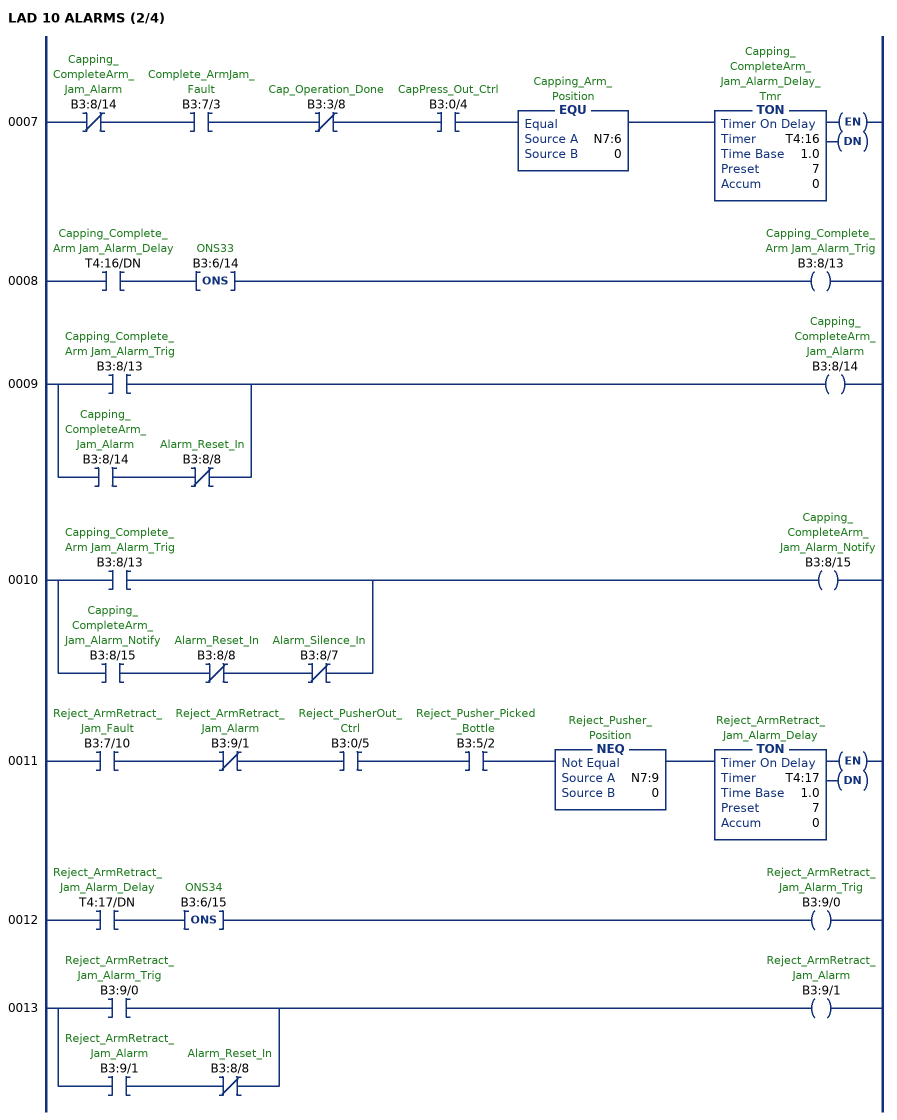
% Rung: 7 %
SOR XIO B3:8/14 XIC B3:7/3 XIO B3:3/8 XIC B3:0/4 EQU N7:6 0 TON T4:16 1.0 7 0 EOR
%   B3:8/14  "Capping_CompleteArm_ Jam_Alarm" %
%   B3:7/3  "Complete_ArmJam_ Fault" %
%   B3:3/8  "Cap_Operation_Done" %
%   B3:0/4  "CapPress_Out_Ctrl" %
%   N7:6  "Capping_Arm_Position" %
%   T4:16  "Capping_CompleteArm_ Jam_Alarm_Delay_Tmr" %
% Rung: 8 %
SOR XIC T4:16/DN ONS B3:6/14 OTE B3:8/13 EOR
%   T4:16/DN  "Capping_Complete_Arm Jam_Alarm_Delay" %
%   B3:6/14  "ONS33" %
%   B3:8/13  "Capping_Complete_Arm Jam_Alarm_Trig" %
% Rung: 9 %
SOR BST XIC B3:8/13 NXB XIC B3:8/14 XIO B3:8/8 BND OTE B3:8/14 EOR
%   B3:8/13  "Capping_Complete_Arm Jam_Alarm_Trig" %
%   B3:8/14  "Capping_CompleteArm_ Jam_Alarm" %
%   B3:8/8  "Alarm_Reset_In" %
% Rung: 10 %
SOR BST XIC B3:8/13 NXB XIC B3:8/15 XIO B3:8/8 XIO B3:8/7 BND OTE B3:8/15 EOR
%   B3:8/13  "Capping_Complete_Arm Jam_Alarm_Trig" %
%   B3:8/15  "Capping_CompleteArm_ Jam_Alarm_Notify" %
%   B3:8/8  "Alarm_Reset_In" %
%   B3:8/7  "Alarm_Silence_In" %
% Rung: 11 %
SOR XIC B3:7/10 XIO B3:9/1 XIC B3:0/5 XIC B3:5/2 NEQ N7:9 0 TON T4:17 1.0 7 0 EOR
%   B3:7/10  "Reject_ArmRetract_ Jam_Fault" %
%   B3:9/1  "Reject_ArmRetract_ Jam_Alarm" %
%   B3:0/5  "Reject_PusherOut_ Ctrl" %
%   B3:5/2  "Reject_Pusher_Picked _Bottle" %
%   N7:9  "Reject_Pusher_ Position" %
%   T4:17  "Reject_ArmRetract_ Jam_Alarm_Delay" %
% Rung: 12 %
SOR XIC T4:17/DN ONS B3:6/15 OTE B3:9/0 EOR
%   T4:17  "Reject_ArmRetract_ Jam_Alarm_Delay" %
%   B3:6/15  "ONS34" %
%   B3:9/0  "Reject_ArmRetract_ Jam_Alarm_Trig" %
% Rung: 13 %
SOR BST XIC B3:9/0 NXB XIC B3:9/1 XIO B3:8/8 BND OTE B3:9/1 EOR
%   B3:9/0  "Reject_ArmRetract_ Jam_Alarm_Trig" %
%   B3:9/1  "Reject_ArmRetract_ Jam_Alarm" %
%   B3:8/8  "Alarm_Reset_In" %

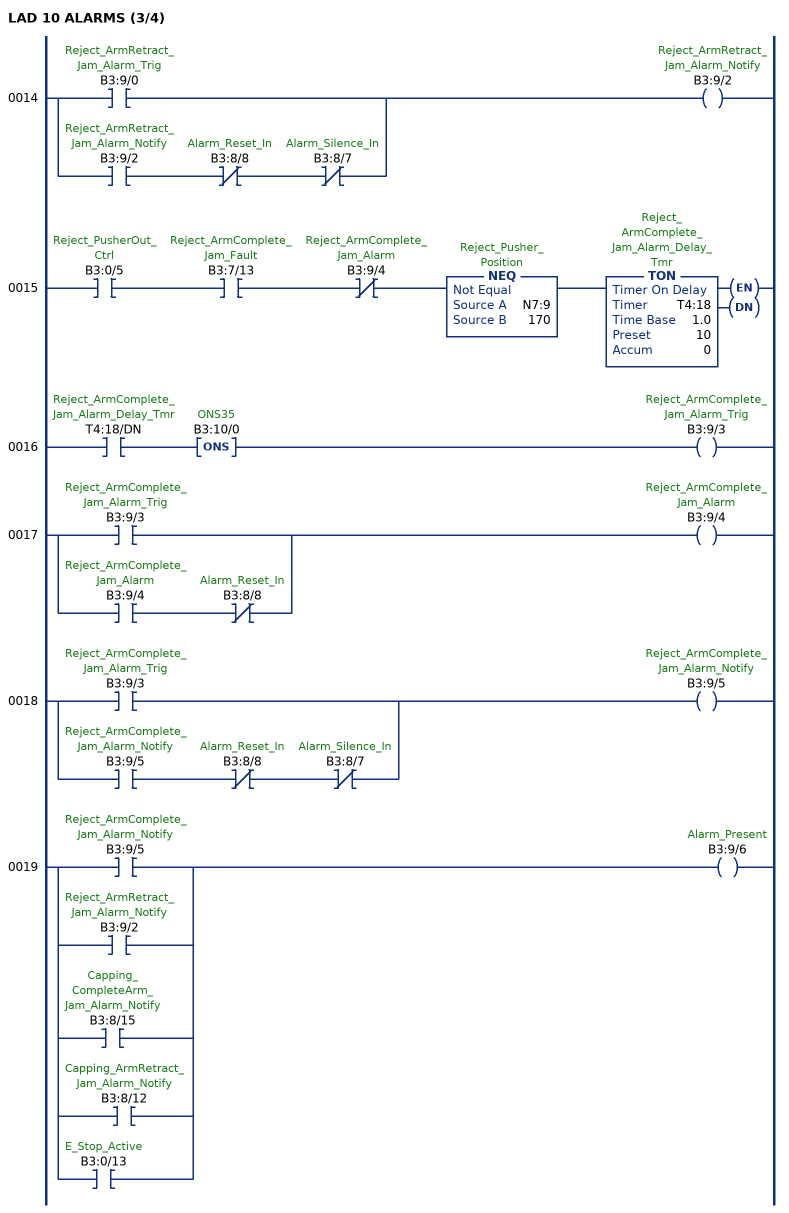
% Rung: 14 %
SOR BST XIC B3:9/0 NXB XIC B3:9/2 XIO B3:8/8 XIO B3:8/7 BND OTE B3:9/2 EOR
%   B3:9/0  "Reject_ArmRetract_ Jam_Alarm_Trig" %
%   B3:9/2  "Reject_ArmRetract_ Jam_Alarm_Notify" %
%   B3:8/8  "Alarm_Reset_In" %
%   B3:8/7  "Alarm_Silence_In" %
% Rung: 15 %
SOR XIC B3:0/5 XIC B3:7/13 XIO B3:9/4 NEQ N7:9 170 TON T4:18 1.0 10 0 EOR
%   B3:0/5  "Reject_PusherOut_ Ctrl" %
%   B3:7/13  "Reject_ArmComplete_ Jam_Fault" %
%   B3:9/4  "Reject_ArmComplete_ Jam_Alarm" %
%   N7:9  "Reject_Pusher_ Position" %
%   T4:18  "Reject_ArmComplete_ Jam_Alarm_Delay_Tmr" %
% Rung: 16 %
SOR XIC T4:18/DN ONS B3:10/0 OTE B3:9/3 EOR
%   T4:18  "Reject_ArmComplete_ Jam_Alarm_Delay_Tmr" %
%   B3:10/0  "ONS35" %
%   B3:9/3  "Reject_ArmComplete_ Jam_Alarm_Trig" %
% Rung: 17 %
SOR BST XIC B3:9/3 NXB XIC B3:9/4 XIO B3:8/8 BND OTE B3:9/4 EOR
%   B3:9/3  "Reject_ArmComplete_ Jam_Alarm_Trig" %
%   B3:9/4  "Reject_ArmComplete_ Jam_Alarm" %
%   B3:8/8  "Alarm_Reset_In" %
% Rung: 18 %
SOR BST XIC B3:9/3 NXB XIC B3:9/5 XIO B3:8/8 XIO B3:8/7 BND OTE B3:9/5 EOR
%   B3:9/3  "Reject_ArmComplete_ Jam_Alarm_Trig" %
%   B3:9/5  "Reject_ArmComplete_ Jam_Alarm_Notify" %
%   B3:8/8  "Alarm_Reset_In" %
%   B3:8/7  "Alarm_Silence_In" %
% Rung: 19 %
SOR BST XIC B3:9/5 NXB XIC B3:9/2 NXB XIC B3:8/15 NXB XIC B3:8/12 NXB XIC B3:0/13 BND OTE B3:9/6 EOR
%   B3:9/5  "Reject_ArmComplete_ Jam_Alarm_Notify" %
%   B3:9/2  "Reject_ArmRetract_ Jam_Alarm_Notify" %
%   B3:8/15  "Capping_CompleteArm_ Jam_Alarm_Notify" %
%   B3:8/12  "Capping_ArmRetract_ Jam_Alarm_Notify" %
%   B3:0/13  "E_Stop_Active" %
%   B3:9/6  "Alarm_Present" %

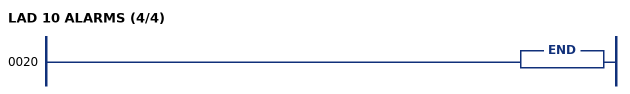
% Rung: 20 %
SOR END EOR

OTHER DOCUMENTED ADDRESSES
  B3:1/8  "AlarmHorn_Trig_Ctrl"
  B3:1/9  "AlarmHorn_Intrpt_Ctr l"
  B3:1/10  "FILL MODE 0 = INCOMPLETE 1 = COMPLETE"
  B3:1/11  "CAPPING MODE 0 = INCOMPLETE 1 = COMPLETE"
  B3:1/12  "SORTING_MODE 0 = INCOMPLETE 1 = COMPLETE"
  B3:1/13  "CAP PRESENT FAULT MODE 0 = CAP PRESENT 1 = CAP ABSENT"
  B3:1/14  "SORTING MODE 0= INCOMPLETE 1 = COMPLETE"
  B3:1/15  "To Packing"
  B3:2/0  "Cycle Complete"
  B3:2/8  "Fill_Station_Bottle_ Present_Trig"
  B3:2/9  "FillStation_Bottle_p resnet_Intrupt"
  B3:3/15  "Bottle Present"
  B3:4/3  "ONS4"
  B3:4/4  "ONS5"
  B3:4/7  "ONS8"
  B3:4/9  "ONS10"
  B3:4/10  "ONS11"
  B3:4/12  "ONS13"
  B3:4/15  "ONS16"
  B3:5/1  "Reject Pusher Move Trig"
  B3:6/0  "ONS17"
  B3:6/7  "ONS24"
  B3:8/4  "Leak_Bottle_Fault_ Alarm_Notify"
  B3:8/9  "Retract_Trig"
  B3:10/1  "ONS36"
  B3:10/3  "ONS37"
  B3:10/5  "ONS38"
  I:0.0/0  "System_Start_PB"
  I:0.0/1  "System Stop PB"
  I:0.0/2  "E_STOP PB"
  I:1.1  "FillLevel_Sensor"
  I:2.0/0  "System_Start_PB"
  I:2.0/1  "System_Stop_PB"
  I:2.0/2  "CapPress_Home_Sensor"
  I:2.0/6  "E_STOP_PB"
  N7:7  "CAP FAULT MOODE"
  N7:8  "Bottle Present"
  N7:19  "BOTTLES PASSED * 3600"
  N7:23  "Bottle_Positioned"
  O:0.0/0  "InfeedConv_Out"
  O:0.0/1  "FillValve_Out"
  T4:0  "Bottle_Arriving_At_ Fill_Station_Delay"
  T4:0/DN  "Bottle_Arrived_Fill_ Station"
  T4:3/EN  "Timer Hold In"
  T4:4  "Capping arm Move delay"
  T4:4/DN  "Capping_Arm_Movement _Inc_Delay"
  T4:6  "Outfeed_Run_Timer"
  T4:6/DN  "Outfed Intrrupt Signal"
  T4:9  "CAPPING TO SORTING MODE DELAY"
  T4:9/DN  "CAPING TO SORTING TRIG"
  T4:12  "Caping Arm Jam Alarm Delay"

COMMENTS NOT ATTACHED TO A CURRENT RUNG
  O:0.0/0: DIGITAL OUTPUTS
  T4:4: SORTING MODE - Sensor Value
  T4:6: Sorting Mode - Packing Mode
  T4:5: Sorting Mode - Rejection Mode

DATA TABLE (non-zero values as saved)
DATA T4
% .PRE .ACC %
% T4:0 % 3 0
% T4:1 % 1 0
% T4:2 % 1 0
% T4:3 % 1 0
% T4:4 % 10 0
% T4:5 % 1 0
% T4:6 % 2 0
% T4:7 % 10 0
% T4:8 % 10 0
% T4:10 % 10 0
% T4:11 % 1 0
% T4:13 % 1 0
% T4:14 % 5 0
% T4:15 % 7 0
% T4:16 % 7 0
% T4:17 % 7 0
% T4:18 % 10 0
% T4:19 % 5 0
% T4:20 % 5 0
